FUNCTION_BLOCK FB_IntFilter
VAR_INPUT
	ValueIn: INT := 0;
	Cycles: INT;
END_VAR
VAR_OUTPUT
	ValueOut: INT;
END_VAR
VAR
	CycleCounter: INT := 0;
	ValueSum: REAL := 0;
	ValueAverage: INT := 0;
	LoopReset: INT;
END_VAR

//CycleCounter := CycleCounter + 1;

IF CycleCounter < Cycles THEN
	ValueSum := ValueSum + INT_TO_REAL(ValueIn) ;
	CycleCounter := CycleCounter + 1;
ELSE
	ValueAverage := REAL_TO_INT(ValueSum / INT_TO_REAL(Cycles)) ;
	ValueOut := ValueAverage;
	ValueSum := 0 ;
	CycleCounter := 0 ;
END_IF

END_FUNCTION_BLOCK

(* stored: Version 1.1.0.1, ProductVersion 3.1.4024.12
   POU FB_IntFilter: Id {b700a9fa-6cfb-45bd-ab7f-f0d55b8c7cc3}, SpecialFunc None *)
